(*
SPDX-FileCopyrightText: © 2026 Oleksandr Tiutyk <trofimich@gmail.com>
SPDX-License-Identifier: MIT
License: https://opensource.org/license/mit
*)

{attribute 'qualified_only'}
{attribute 'strict'}
{attribute 'to_string'}
TYPE ERROR_SEVERITY :
(
	ERROR := 0,
	CRITICAL
);
END_TYPE

(* stored: Version 1.1.0.1
   DUT ERROR_SEVERITY: Id {232be12d-183d-4200-abbc-93d81956178a} *)
